ABB RAPID module: Module1.mod

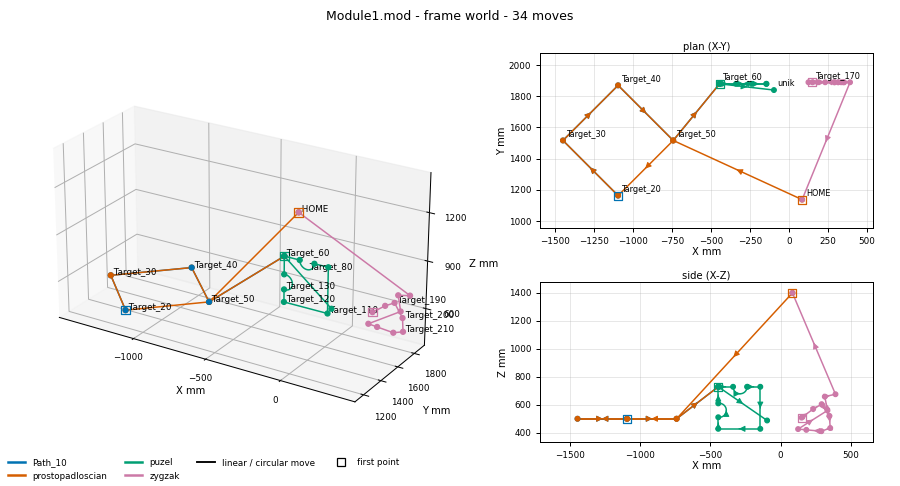
[picture p0: tool path of Module1.mod in frame world, 34 of 34 moves have a stored position in this frame; points joined in program order, loops and branches not executed]
MODULE Module1
	CONST robtarget Target_20:=[[-1095.097661644,1163.266131464,500],[0,0.923879533,0.382683432,0],[1,-2,0,1],[9E+09,9E+09,9E+09,9E+09,9E+09,9E+09]];
	CONST robtarget Target_30:=[[-1448.651052237,1516.819522058,500],[0,0.923879533,0.382683432,0],[1,-2,0,1],[9E+09,9E+09,9E+09,9E+09,9E+09,9E+09]];
	CONST robtarget Target_40:=[[-1095.097661644,1870.372912651,500],[0,0.923879533,0.382683432,0],[1,-2,0,1],[9E+09,9E+09,9E+09,9E+09,9E+09,9E+09]];
	CONST robtarget Target_50:=[[-741.544271051,1516.819522058,500],[0,0.923879533,0.382683432,0],[1,-2,0,1],[9E+09,9E+09,9E+09,9E+09,9E+09,9E+09]];
	CONST robtarget Target_60:=[[-444.296598994,1880,728.176467536],[0.707106781,-0.707106781,0,0],[1,0,-2,1],[9E+09,9E+09,9E+09,9E+09,9E+09,9E+09]];
	CONST robtarget Target_10:=[[-741.544271051,1516.819522058,500],[0,0.923879533,0.382683432,0],[1,-2,0,1],[9E+09,9E+09,9E+09,9E+09,9E+09,9E+09]];
	CONST robtarget Target_70:=[[-338.609598994,1880,728.176467536],[0.707106781,-0.707106781,0,0],[1,-1,-1,1],[9E+09,9E+09,9E+09,9E+09,9E+09,9E+09]];
	CONST robtarget Target_80:=[[-288.609598994,1880,678.176467536],[0.707106781,-0.707106781,0,0],[1,-1,-1,1],[9E+09,9E+09,9E+09,9E+09,9E+09,9E+09]];
	CONST robtarget Target_90:=[[-238.609598994,1880,728.176467536],[0.707106781,-0.707106781,0,0],[1,-1,-1,1],[9E+09,9E+09,9E+09,9E+09,9E+09,9E+09]];
	CONST robtarget Target_100:=[[-144.296598994,1880,728.176467536],[0.707106781,-0.707106781,0,0],[1,-1,-1,1],[9E+09,9E+09,9E+09,9E+09,9E+09,9E+09]];
	CONST robtarget Target_110:=[[-144.296598994,1880,428.176467536],[0.707106781,-0.707106781,0,0],[1,-1,-1,1],[9E+09,9E+09,9E+09,9E+09,9E+09,9E+09]];
	CONST robtarget Target_120:=[[-444.296598994,1880,428.176467536],[0.707106781,-0.707106781,0,0],[1,0,-2,1],[9E+09,9E+09,9E+09,9E+09,9E+09,9E+09]];
	CONST robtarget Target_130:=[[-444.296598994,1880,510.750512977],[0.707106781,-0.707106781,0,0],[1,0,-2,1],[9E+09,9E+09,9E+09,9E+09,9E+09,9E+09]];
	CONST robtarget Target_140:=[[-386.8491628,1880,560.192759023],[0.707106781,-0.707106781,0,0],[1,-1,-1,1],[9E+09,9E+09,9E+09,9E+09,9E+09,9E+09]];
	CONST robtarget Target_150:=[[-444.296598994,1880,609.63500507],[0.705132066,-0.705132066,-0.052808804,-0.052808804],[1,0,-2,1],[9E+09,9E+09,9E+09,9E+09,9E+09,9E+09]];
	CONST robtarget Target_160:=[[-444.296598994,1880,728.176467536],[0.707106781,-0.707106781,0,0],[1,0,-2,1],[9E+09,9E+09,9E+09,9E+09,9E+09,9E+09]];
	CONST robtarget Target_170:=[[150.794,1890,507.946],[0.670707042,-0.670707042,-0.223946564,-0.223946564],[0,-1,-2,1],[9E+09,9E+09,9E+09,9E+09,9E+09,9E+09]];
	CONST robtarget Target_180:=[[232.858,1890,569.624],[0.670707042,-0.670707042,-0.223946564,-0.223946564],[0,-1,-2,1],[9E+09,9E+09,9E+09,9E+09,9E+09,9E+09]];
	CONST robtarget Target_190:=[[293.567,1890,604.039],[0.6837289,-0.6837289,-0.180318582,-0.180318582],[0,-1,-2,1],[9E+09,9E+09,9E+09,9E+09,9E+09,9E+09]];
	CONST robtarget Target_200:=[[348.655,1890,520.673],[0.677182322,-0.677182322,-0.203529119,-0.203529119],[0,-1,-2,1],[9E+09,9E+09,9E+09,9E+09,9E+09,9E+09]];
	CONST robtarget Target_210:=[[354.711,1890,433.624],[0.706680401,-0.706680401,-0.02455221,-0.02455221],[0,-1,-1,1],[9E+09,9E+09,9E+09,9E+09,9E+09,9E+09]];
	CONST robtarget Target_220:=[[291.616,1890,411.171],[0.696800555,-0.696800555,-0.120287098,-0.120287098],[0,-1,-2,1],[9E+09,9E+09,9E+09,9E+09,9E+09,9E+09]];
	CONST robtarget Target_230:=[[184.066,1890,420.799],[0.706402312,-0.706402312,0.031555878,0.031555878],[0,-1,-1,1],[9E+09,9E+09,9E+09,9E+09,9E+09,9E+09]];
	CONST robtarget Target_240:=[[125.576,1890,426.313],[0.706326013,-0.706326013,0.033219923,0.033219923],[0,-1,-1,1],[9E+09,9E+09,9E+09,9E+09,9E+09,9E+09]];
	CONST robtarget Target_250:=[[335.11,1890,559.284],[0.702836094,-0.702836094,0.077597845,0.077597845],[0,-1,-1,1],[9E+09,9E+09,9E+09,9E+09,9E+09,9E+09]];
	CONST robtarget Target_260:=[[315.857,1890,657.938],[0.703826001,-0.703826001,-0.06803646,-0.06803646],[0,-1,-1,1],[9E+09,9E+09,9E+09,9E+09,9E+09,9E+09]];
	CONST robtarget Target_270:=[[392.275,1890,674.977],[0.702857034,-0.702857034,-0.077407942,-0.077407942],[0,-1,-1,1],[9E+09,9E+09,9E+09,9E+09,9E+09,9E+09]];
    CONST robtarget HOME:=[[84.951039934,1137.529040422,1397.771840852],[0.00939952,0.969365782,0.215763318,0.116994958],[0,-2,0,1],[9E+09,9E+09,9E+09,9E+09,9E+09,9E+09]];
    CONST robtarget unik:=[[-95.717892828,1840.102968068,487.702541424],[0.670707014,-0.670706715,-0.223947139,-0.223947052],[1,-1,-2,1],[9E+09,9E+09,9E+09,9E+09,9E+09,9E+09]];
    !***********************************************************
    !
    ! Module:  Module1
    !
    ! Description:
    !   <Insert description here>
    !
    ! Author: festo
    !
    ! Version: 1.0
    !
    !***********************************************************


    !***********************************************************
    !
    ! Procedure main
    !
    !   This is the entry point of your program
    !
    !***********************************************************
    PROC main()
        prostopadloscian;
        puzel;
        zygzak;
    ENDPROC
	PROC Path_10()
	    MoveL Target_20,v1000,z100,dupsko_bonczura\WObj:=wobj0;
	    MoveL Target_30,v1000,z100,dupsko_bonczura\WObj:=wobj0;
	    MoveL Target_40,v1000,z100,dupsko_bonczura\WObj:=wobj0;
	    MoveL Target_50,v1000,z100,dupsko_bonczura\WObj:=wobj0;
	    MoveL Target_60,v1000,z100,dupsko_bonczura\WObj:=wobj0;
	ENDPROC
	PROC prostopadloscian()
	    MoveL HOME,v1000,z100,dupsko_bonczura\WObj:=wobj0;
	    MoveL Target_10,v1000,fine,dupsko_bonczura\WObj:=wobj0;
	    MoveL Target_20,v150,fine,dupsko_bonczura\WObj:=wobj0;
	    MoveL Target_30,v150,fine,dupsko_bonczura\WObj:=wobj0;
	    MoveL Target_40,v150,fine,dupsko_bonczura\WObj:=wobj0;
	    MoveL Target_50,v150,fine,dupsko_bonczura\WObj:=wobj0;
	    MoveL Target_60,v1000,fine,dupsko_bonczura\WObj:=wobj0;
	ENDPROC
	PROC puzel()
	    MoveL Target_60,v1000,fine,dupsko_bonczura\WObj:=wobj0;
	    MoveL Target_70,v150,fine,dupsko_bonczura\WObj:=wobj0;
	    MoveC Target_80,Target_90,v150,fine,dupsko_bonczura\WObj:=wobj0;
	    MoveL Target_100,v150,fine,dupsko_bonczura\WObj:=wobj0;
	    MoveL Target_110,v150,fine,dupsko_bonczura\WObj:=wobj0;
	    MoveL Target_120,v150,fine,dupsko_bonczura\WObj:=wobj0;
	    MoveL Target_130,v150,fine,dupsko_bonczura\WObj:=wobj0;
	    MoveC Target_140,Target_150,v150,fine,dupsko_bonczura\WObj:=wobj0;
	    MoveL Target_160,v150,fine,dupsko_bonczura\WObj:=wobj0;
        MoveL unik,v500,z100,dupsko_bonczura\WObj:=wobj0;
	ENDPROC
	PROC zygzak()
	    MoveL Target_170,v1000,z100,dupsko_bonczura\WObj:=wobj0;
	    MoveL Target_180,v150,z100,dupsko_bonczura\WObj:=wobj0;
	    MoveL Target_190,v150,z100,dupsko_bonczura\WObj:=wobj0;
	    MoveL Target_200,v150,z100,dupsko_bonczura\WObj:=wobj0;
	    MoveL Target_210,v150,z100,dupsko_bonczura\WObj:=wobj0;
	    MoveL Target_220,v150,z100,dupsko_bonczura\WObj:=wobj0;
	    MoveL Target_230,v150,z100,dupsko_bonczura\WObj:=wobj0;
	    MoveL Target_240,v150,z100,dupsko_bonczura\WObj:=wobj0;
	    MoveL Target_250,v150,z100,dupsko_bonczura\WObj:=wobj0;
	    MoveL Target_260,v150,z100,dupsko_bonczura\WObj:=wobj0;
	    MoveL Target_270,v150,z100,dupsko_bonczura\WObj:=wobj0;
        MoveL HOME,v1000,fine,dupsko_bonczura\WObj:=wobj0;
	ENDPROC
ENDMODULE
